(* CoDeSys 2.3.9.52 project: BRE.pro *)
(* Libraries: Standard.lib 20.5.14 09:13:26, Iecsfc.lib 30.1.13 14:05:12, SYSLIBCALLBACK.LIB 30.1.13 14:05:12, C:\Program Files (x86)\WAGO Software\CoDeSys V2.3\Targets\WAGO\Libraries\oscat\oscat_building_100.lib 27.1.16 15:07:45, C:\Program Files (x86)\WAGO Software\CoDeSys V2.3\Targets\WAGO\Libraries\Building\English\Building_common.lib 1.2.07 14:25:42 *)

(* PLC configuration (modules and I/O channels)
K-Bus [K_Bus] node 0, in %IB0 out %QB0 {KbusBusMode = 1; KbusCycleTime = 10000; KbusThreadPriority = 0; KbusSetOutputsToZeroOnApplicationStop = 1}
IEC60870-5-Konfig [IEC60870_Konfig] node 1, in %IB10000 out %QB10000 {IEC870_tAFZ_Kurz = t#500ms; IEC870_tAFZ_Lang = t#5s; IEC870_tAFZ_Default = t#2s; IEC870_nMaxTLGBufferSize = 32; IEC870_xUseSNTP = 1; IEC870_byTaskPrio = 21; IEC870_tTaskTime = t#20ms; IEC870_byTaskPrio = 22; IEC870_tTaskTime = t#20ms; IEC870_byTaskPrio = 23; IEC870_tTaskTime = t#20ms; IEC870_byTaskPrio = 24; IEC870_tTaskTime = t#20ms; IEC870_byVarGenMode = 1; IEC870_sSelSprache = DEUTSCH; IEC870_sTargetTyp = 758-8xx; IEC870_sUsedLib = Standard.LIB; IEC870_sUsedLib = SysLibCallback.LIB; IEC870_sUsedLib = SysLibRtc.LIB; IEC870_sUsedLib = SysLibSockets.LIB; IEC870_sUsedLib = SysLibMem.LIB; IEC870_sUsedLib = SysLibTime.LIB; IEC870_sUsedLib = SysLibSem.LIB; IEC870_sUsedLib = SysLibCom.LIB; IEC870_sInputAdr640 = %IB0; IEC870_sOutputAdr640 = %QB0; IEC870_UsedInfoObjFB_V2 = TRUE; IEC870_NTP_ServerAdress = 192.53.103.108; IEC870_NTP_RequestResponseTime = t#50ms; IEC870_NTP_UpdateIntervall = 60; IEC870_NTP_WatchdogTime = 10; IEC870_sUsedLib = SerComm.LIB; IEC870_sUsedLib = WagoLibEthernet_01.lib; IEC870_sUsedLib = WagoLibSntp.LIB; IEC870_sUsedLib = WagoLibNTP.LIB; IEC870_sUsedLib = WagoLibPing.lib; IEC870_sUsedLib = WagoLib60870Base.lib; IEC870_sUsedLib = WagoLib60870Slave.lib; IEC870_sUsedLib = WagoLib60870Master.lib; gsiIEC870_CLOCK_TimeZone = 0; gnIEC870_CLOCK_DST_Mode = 0; IEC870_xZW_SendSpoantan = 0; IEC870_diTimeOutC_Objs = 1000; IEC870_diHistBufferSize = 16; IEC870_xEnableGaForCpObj = 1; IEC870_byParameter = 0; IEC870_diParameter = 0; IEC870_diParameter = 0; IEC870_diParameter = 0; IEC870_byParameter = 0; IEC870_byParameter = 0; IEC870_byParameter = 0; IEC870_sParameter = 0; IEC870_sParameter = 0; IEC870_sParameter = 0}
Modbus variables [PFC200MODBUS] node 2, in %IB0 out %QB0 {PlcStopBehaviour = 1; FiledbusErrorBehaviour = 1; TcpOperation = 1; TcpPort = 502; TcpTimeout = 600; UdpOperation = 1; UdpPort = 502; RtuOperation = 0; NodeId = 1; ResponseTimeout = 100; Interface = 0; Baud = 115200; StopBits = 1; Parity = 1; FlowCtrl = 0; PhysInterface = 0}
IEC61850-Konfig [IEC61850_Konfig] node 3, in %IB10000 out %QB10000 {IEC61850_sSelSprache = DEUTSCH; IEC61850_sTargetTyp = 758-8xx}
DNP3-Konfig [DNP3_Konfig] node 4, in %IB10000 out %QB10000 {IEC61850_sSelSprache = DEUTSCH; IEC61850_sTargetTyp = 758-8xx}
Modbus-Master [MB_MASTER] node 5, in %IB0 out %QB0
*)

(* POU PLC_PRG, CFC *)
PROGRAM PLC_PRG
VAR
	time_day: BOOL;
	season: BOOL;
	presence_room_08: BOOL;
	room_08HVAC_mode: BOOL;
	g_security_mode: BOOL;
	room_08switch_01: BOOL;
	lg_02_actor_fb: BOOL;
	room_08_movement_sensor: BOOL;
	g_day_night: BOOL;
	cmd_room_08_lg_01: BOOL;
	room_08_blind_pos_fb: BOOL;
	room_08_light_level: BOOL;
END_VAR
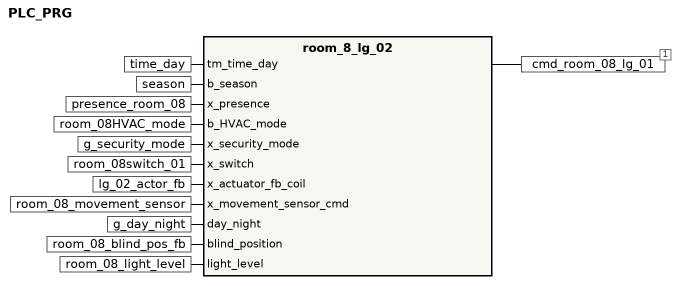
_CFC_ (* Continuous Function Chart, elements in execution order *)
#0 room_8_lg_02(tm_time_day: time_day, b_season: season, x_presence: presence_room_08, b_HVAC_mode: room_08HVAC_mode, x_security_mode: g_security_mode, x_switch: room_08switch_01, x_actuator_fb_coil: lg_02_actor_fb, x_movement_sensor_cmd: room_08_movement_sensor, day_night: g_day_night, blind_position: room_08_blind_pos_fb, light_level: room_08_light_level)
#1 cmd_room_08_lg_01 <= #0
_END_CFC_
(* the same logic as Structured Text *)
cmd_room_08_lg_01 := room_8_lg_02(tm_time_day := time_day, b_season := season, x_presence := presence_room_08, b_HVAC_mode := room_08HVAC_mode, x_security_mode := g_security_mode, x_switch := room_08switch_01, x_actuator_fb_coil := lg_02_actor_fb, x_movement_sensor_cmd := room_08_movement_sensor, day_night := g_day_night, blind_position := room_08_blind_pos_fb, light_level := room_08_light_level);
END_PROGRAM

(* POU room_8_lg_02, CFC *)
FUNCTION room_8_lg_02 : BOOL

VAR_INPUT
	tm_time_day: STRING;
	b_season: WORD;
	x_presence:BOOL;
	b_HVAC_mode :WORD;
	x_security_mode :BOOL;
	x_switch: BOOL;
	x_actuator_fb_coil: BOOL;
	x_movement_sensor_cmd: BOOL;
	day_night:BOOL;
	blind_position: BYTE;
	light_level:WORD;




END_VAR
VAR
	CLICK: CLICK;
	rtrig01: R_TRIG;
END_VAR
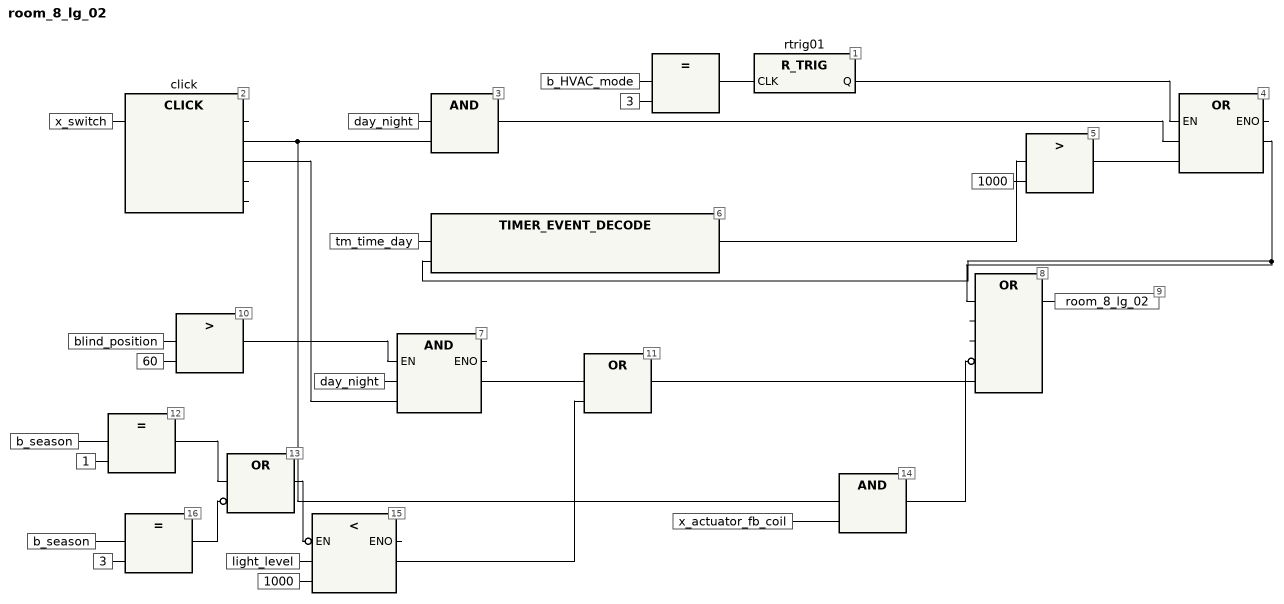
_CFC_ (* Continuous Function Chart, elements in execution order *)
#0 =(b_HVAC_mode, 3)
#1 rtrig01:R_TRIG(CLK: #0)
#2 click:CLICK(x_switch)
#3 AND(day_night, #2.out 2)
#4 OR(EN: #1.Q, #3, #5)
#5 >(#6, 1000)
#6 TIMER_EVENT_DECODE(tm_time_day, #4)
#7 AND(EN: #10, day_night, #2.out 3)
#8 OR(#4, -, -, NOT #14, #11)
#9 room_8_lg_02 <= #8
#10 >(blind_position, 60)
#11 OR(#7, #15)
#12 =(b_season, 1)
#13 OR(#12, NOT #16)
#14 AND(#2.out 2, x_actuator_fb_coil)
#15 <(EN: NOT #13, light_level, 1000)
#16 =(b_season, 3)
_END_CFC_
END_FUNCTION
